PROGRAM MAIN
VAR
	{region 'State Machine Variables'}
	// State of the state machine
	nState 			: INT;
	// Control Variables
	bStart, bHalt 	: BOOL;
	{endregion}
	
	{region 'NC Variables'}
	// Axis Control Ref
	Axis			: ARRAY[1..3] OF Axis_Ref;
	// Axis Power Block
	mcPower 		: ARRAY[1..3] OF MC_Power;
	// Axis Move Absolute Block
	mcMoveAbs 		: MC_MoveAbsolute;
	// Absolute Position
	fPosition 		: LREAL := POSITION_A;
	// Gear-In Function Block
	mcGearIn 		: MC_GearIn;
	// External Setpoint Gen Enable
	mcExtSpEnable 	: MC_ExtSetPointGenEnable;
	// Gen Feed Direction
	nDirection		: DINT;
	{endregion}

	{region  'General System Variables'}
	// Loop Iterator
	I_itr			: INT;
	// Random Position
	Random			: DRAND;
	// Dwell Timer
	Dwell 			: TON;
	{endregion}
END_VAR
VAR CONSTANT
	{region  'Position Constants'}
	// Position A Setpoint
	POSITION_A 		: LREAL := -5000;
	// Position B Setpoint
	POSITION_B 		: LREAL := 5000;
	{endregion}
END_VAR

// Simple NC State Machine

CASE nState OF
	{region 'Start of State Machine'}
	0:	// Start the state machine
		IF bStart THEN
			bStart := FALSE;
			nState := nState + 10;
		END_IF
	{endregion}
	
	{region 'Axes Power Section'}
	10: // Power on the axis
		FOR I_itr := 1 TO 3 DO
			mcPower[I_itr](Axis := Axis[I_itr], Enable := TRUE, Enable_Positive := TRUE, Enable_Negative := TRUE, Override := 100.0);
		END_FOR
		nState := nState + 10;
	
	20: // Check all axis are enabled
		FOR I_itr := 1 TO 3 DO
			// Check if motor is enabled
			IF NOT mcPower[I_itr].Status THEN
				// Return to power state, or reset state if you have one
				// At the end of this state we add 10, so to return to 10 we need to subtract 20
				nState := nState - 20;
				EXIT;
			END_IF
		END_FOR
		nState := nState + 10;
	{endregion}
		 
	{region 'Exercise 2 - GearIn Function'}	
	30: (*
		**	Exercise 2 - Gear-In Axis 2 to Axis 1
		*)
		mcGearIn(Master:= Axis[1], Slave:= Axis[2], Execute:= TRUE, RatioNumerator:= 0.5, RatioDenominator:= 1);
		IF mcGearIn.InGear THEN
			mcGearIn(Master:= Axis[1], Slave:= Axis[2], Execute:= FALSE, RatioNumerator:= 0.5, RatioDenominator:= 1);
			nState := nState + 10;
		END_IF
	{endregion}
	
	{region 'Exercise 3 - External Setpoint'}		 
	40: (*
		**	Exercise 3 - Enable External Setpoint Generator for Axis 3
		*)
		mcExtSpEnable(Axis:= Axis[3], Execute:= TRUE, Position:= 0, PositionType:= POSITIONTYPE_ABSOLUTE);
		IF mcExtSpEnable.Done THEN
			mcExtSpEnable(Axis:= Axis[3], Execute:= FALSE, Position:= 0, PositionType:= POSITIONTYPE_ABSOLUTE);
			nState := nState + 10;
		END_IF
	{endregion}	
		 
	{region 'Exercise 1 - Reversing Sequence'}		
	50: (*
		** Exercise 1 - Execute an absolute move on Axis 1 and wait here until done
		*)
		// Execute move to Position A
		mcMoveAbs(Axis:= Axis[1], Execute:= TRUE, Position:= fPosition, Velocity := 1000, Acceleration := 2000, Deceleration := 2000, Jerk := 5000);
		// Check if move is complete
		IF mcMoveAbs.Done THEN
			mcMoveAbs(Axis:= Axis[1], Execute:= FALSE);
			nState := nState + 10;
		END_IF
		
	60: (*
		** Exercise 1 - Call a dwell timer, wait here until time is elapsed
		*)
		Dwell(IN:= TRUE, PT:= T#1S);
		IF Dwell.Q THEN
			Dwell(IN:= FALSE, PT:= T#1S);
			nState := nState + 10;
		END_IF
		
		
	70: (*
		** Exercise 1 - Check what position was last issued, and command a new one
		*)
		// Swap the position
		//IF fPosition = POSITION_A THEN
		//	fPosition := POSITION_B;
		//ELSE
		//	fPosition := POSITION_A;
		//END_IF
		Random(Seed:= 1, Num=> fPosition);
		IF Axis[1].NcToPlc.ActPos > 0 THEN
			fPosition := fPosition * -5000.0;
		ELSE
			fPosition := fPosition * 5000.0;
		END_IF	
		nState := nState + 10;
	{endregion}
		
	{region 'End of State Machine'}
	80:
		// Check if continuous loop, or return to 0
		IF bHalt THEN
			bHalt := TRUE;
			nState := 0;
		ELSE
			nState := nState - 30;
		END_IF
	{endregion}		
END_CASE
{region 'Exercise 3 - External Setpoint'}	
(* 
** Exercise 3 - External Setpoint Generator Feed 
*)

// Read the status of Axis 1
Axis[1].ReadStatus();

// Read the direction of Axis 1 and map it to Axis 3
IF Axis[1].Status.PositiveDirection THEN
	nDirection := 1;
ELSIF Axis[1].Status.NegativeDirection THEN
	nDirection := -1;
ELSE
	nDirection := 0;
END_IF

// Call the Setpoint Feed
MC_ExtSetPointGenFeed(Position:= Axis[1].NcToPlc.ActPos, Velocity:= Axis[1].NcToPlc.ActVelo, Acceleration:= Axis[1].NcToPlc.ActAcc, Direction:= nDirection, Axis:= Axis[3]);
{endregion}

END_PROGRAM

(* stored: Version 1.1.0.1, ProductVersion 3.1.4024.12
   POU MAIN: Id {42e41504-19b0-4be3-aee2-d44241402398}, SpecialFunc None *)
